// TIA Portal V17 export
// export: Created 2025-03-07T09:19:06.9362138Z, ExportSetting WithDefaults, DisplayName Totally Integrated Automation Portal, DisplayVersion V17 Update 8, DisplayName TIA Portal Openness, DisplayVersion V17 Update 8, DisplayName TIA Portal Version Control Interface, DisplayVersion V17, DisplayName SINAMICS Startdrive Advanced, DisplayVersion V17 SP2, DisplayName SINAMICS Startdrive G110M, G120, G120C, G120D, G120P, G115D, DisplayVersion V17 SP2, DisplayName SINAMICS Startdrive G130, G150, S120, S150, SINAMICS MV, S210, DisplayVersion V17 SP2, DisplayName STEP 7 Professional, DisplayVersion V17 Update 8, DisplayName SINUMERIK ONE STEP 7 Toolbox, DisplayVersion V17 Update 12, DisplayName SINUMERIK 840D sl STEP 7 Toolbox, DisplayVersion V17 Update 12, DisplayName STEP 7 Safety, DisplayVersion V17 Update 6, DisplayName WinCC Advanced, DisplayVersion V17 Update 8
FUNCTION "FC10100_POWDER_FLOW_SENSOR_MEDICOAT" : Void   // FC10100, LAD
{ S7_Optimized_Access := 'TRUE' }
VERSION : 0.1
// stored: AutoNumber false, IsIECCheckEnabled false, SetENOAutomatically false, UDAEnableTagReadback false
BEGIN

REGION Network 1: UNIT 01
END_REGION

REGION Network 2: LASER HEAD MEDICOAT
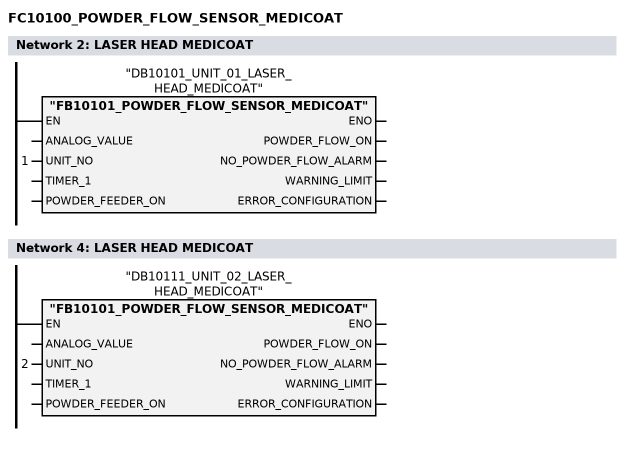
   RUNG wire#powerrail
      "DB10101_UNIT_01_LASER_HEAD_MEDICOAT"(ANALOG_VALUE :=, UNIT_NO := 1, TIMER_1 :=, POWDER_FEEDER_ON :=, POWDER_FLOW_ON =>, NO_POWDER_FLOW_ALARM =>, WARNING_LIMIT =>, ERROR_CONFIGURATION =>)
   END_RUNG
   // the same network as SCL:
   "DB10101_UNIT_01_LASER_HEAD_MEDICOAT"(UNIT_NO := 1);   // "FB10101_POWDER_FLOW_SENSOR_MEDICOAT"
END_REGION

REGION Network 3: UNIT 02
END_REGION

REGION Network 4: LASER HEAD MEDICOAT
   RUNG wire#powerrail
      "DB10111_UNIT_02_LASER_HEAD_MEDICOAT"(ANALOG_VALUE :=, UNIT_NO := 2, TIMER_1 :=, POWDER_FEEDER_ON :=, POWDER_FLOW_ON =>, NO_POWDER_FLOW_ALARM =>, WARNING_LIMIT =>, ERROR_CONFIGURATION =>)
   END_RUNG
   // the same network as SCL:
   "DB10111_UNIT_02_LASER_HEAD_MEDICOAT"(UNIT_NO := 2);   // "FB10101_POWDER_FLOW_SENSOR_MEDICOAT"
END_REGION
END_FUNCTION
